FUNCTION_BLOCK FB_Controller
VAR_INPUT
	fNewRate : REAL;
	bPumpOn : BOOL;
	bPumpOff : BOOL;
END_VAR
VAR
	iPump : I_Pump;
	iAdjustPump : I_AdjustablePump;
	bAdjustable : BOOL;
END_VAR

IF bPumpOn THEN
	IF iPump <> 0 THEN
		iPump.Start();
		IsAdjustable();
		IF bAdjustable THEN
		iAdjustPump.SetFlowRate(fNewRate);
		END_IF
	END_IF
END_IF
IF bPumpOff THEN
	IF iPump <> 0 THEN
		iPump.Stop();
	END_IF
	
END_IF

METHOD FB_init : BOOL
VAR_INPUT
	bInitRetains : BOOL; // if TRUE, the retain variables are initialized (warm start / cold start)
	bInCopyCode : BOOL;  // if TRUE, the instance afterwards gets moved into the copy code (online change)
	_iPump : I_Pump;
END_VAR
iPump := _iPump;
END_METHOD

METHOD IsAdjustable 
VAR_INPUT
END_VAR
bAdjustable := __QUERYINTERFACE(iPump, iAdjustPump);
END_METHOD

END_FUNCTION_BLOCK

(* stored: Version 1.1.0.1, ProductVersion 3.1.4024.16
   POU FB_Controller: Id {a3eb19ff-1505-4bf8-b69d-ca8845e7835d}, SpecialFunc None
   Method FB_init: Id {8a32dfa8-b2d8-4850-95e6-67b3bf47d6ab}
   Method IsAdjustable: Id {8fc6ca95-5c23-4607-b5e9-90871c7b4005} *)
